// TwinCAT 3 PLC project vonhamos_motion
// ProgramVersion: 3.1.4022.7
// libraries:
//   Tc2_Standard, * (Beckhoff Automation GmbH)
//   Tc2_System, * (Beckhoff Automation GmbH)
//   Tc3_Module, * (Beckhoff Automation GmbH)
//   lcls-twincat-motion,1.3.2,SLAC
// project tree:
//   / PlcTask.TcTTO (not stored)
//   POUs/ Main.TcPOU
// real-time tasks:
//   TASK PlcTask: cycle T#10ms, priority 20, ADS port 350
// motion (NC):
//   TASK NC-Task 1 SAF: cycle T#2ms, priority 4, ADS port 501
//   TASK NC-Task 1 SVB: cycle T#10ms, priority 8, ADS port 511
//   AXIS VonHamosY (id 1)
//     OtherSettings: AllowMotionCmdToSlave=true
//     encoder EncType=1
//     drive DrvType=5
//       Analog: ScaleFactorActTorque=0.1
//     controller CtrType=1
//       CtrPara: PriorControlFactor=1
//         Observer: BandWidth=20
// variable links:
//   vonhamos_motion Instance <-> NC-Task 1 SAF/Axes/VonHamosY
//     PlcTask Inputs/Main.M1.Axis.NcToPlc <-> Outputs/ToPlc
//     PlcTask Outputs/Main.M1.Axis.PlcToNc <-> Inputs/FromPlc

// ---- POUs/Main.TcPOU
PROGRAM Main
VAR
	// Motors
	{attribute 'TcLinkTo' := '.bLimitForwardEnable:=TIIB[VonHamosY-EL7041]^STM Status^Status^Digital input 1;
                              .bLimitBackwardEnable:=TIIB[VonHamosY-EL7041]^STM Status^Status^Digital input 2'}
	{attribute 'pytmc' := '
		pv: HXX:VON_HAMOS:MMS:01
	'}
	M1 : DUT_MotionStage; // Y axis

	fbMotionStageM1 : FB_MotionStage;
END_VAR

// Hardware Enable
M1.bHardwareEnable := TRUE;
fbMotionStageM1(stMotionStage:=M1);

END_PROGRAM
